/// \copydoc ZCore.ITestContext
FUNCTION_BLOCK TestContext IMPLEMENTS ITestContext
VAR
  _busy : BOOL;
  _userData : POINTER TO BYTE;
  _assertions : IAssertions;
END_VAR

/// \copydoc ZCore.ITestContext#Assertions
PROPERTY Assertions : IAssertions
GET
Assertions := _assertions;
END_GET
END_PROPERTY

/// \copydoc ZCore.ITestContext#Busy
PROPERTY Busy : BOOL
GET
Busy := _busy;
END_GET
SET
_busy := Busy;
END_SET
END_PROPERTY

METHOD FB_init : BOOL
VAR_INPUT
	bInitRetains : BOOL; // if TRUE, the retain variables are initialized (warm start / cold start)
	bInCopyCode : BOOL;  // if TRUE, the instance afterwards gets moved into the copy code (online change)
  assertions : IAssertions;
END_VAR
END_METHOD

/// \copydoc ZCore.ITestContext#UserData
PROPERTY UserData : POINTER TO BYTE
GET
UserData := _userData;
END_GET
SET
_userData := UserData;
END_SET
END_PROPERTY

END_FUNCTION_BLOCK

(* stored: Version 1.1.0.1, ProductVersion 3.1.4024.12
   POU TestContext: Id {c1aced88-be98-472e-8f3a-706ec0cf984c}, SpecialFunc None
   Property Assertions: Id {2286251f-9ed5-4103-a8b2-a6cfe89617ff}
   Get Get: Id {74ce47ef-885a-41ac-8d77-24d455a1feee}
   Property Busy: Id {3f2ccdca-2f47-4173-8394-b59b5ae1f634}
   Get Get: Id {ceb958e3-d0f3-4809-b2c0-955567b7d4d9}
   Set Set: Id {f5c16378-b380-42d4-9305-3d18205aa5b9}
   Method FB_init: Id {88ac0017-8517-4852-bafc-43b0ca4e0cd4}
   Property UserData: Id {cc2e97fe-2a7f-4bce-8506-d0d6e29333fa}
   Get Get: Id {974fe803-b308-4ab6-8c69-785b8149c931}
   Set Set: Id {61fd05d2-1396-4298-9b45-ecf9ac10c2b6} *)
